// TIA Portal project "Tank_V17" (V17)

(* hardware
DEVICE "S7-1200-Station_1"  S7-1200 Station
   slot 0: "Baugruppenträger_0"  S7-1200 Rack  Rack  V1.0
   slot 1: "PLC_1"  CPU 1214C DC/DC/DC  6ES7 214-1AG40-0XB0  V4.2
   slot 3: "AQ 1x12BIT_1"  AQ1 signal board  6ES7 232-4HA30-0XB0  V1.0
*)

// ===== PLC "PLC_1"  CPU 1214C DC/DC/DC =====

VAR_GLOBAL   // PLC tag table "Standard-Variablentabelle"
   "System_Byte" AT %MB100 : Byte;
   "FirstScan" AT %M100.0 : Bool;
   "DiagStatusUpdate" AT %M100.1 : Bool;
   "AlwaysTRUE" AT %M100.2 : Bool;
   "AlwaysFALSE" AT %M100.3 : Bool;
   "Clock_Byte" AT %MB110 : Byte;
   "Clock_10Hz" AT %M110.0 : Bool;
   "Clock_5Hz" AT %M110.1 : Bool;
   "Clock_2.5Hz" AT %M110.2 : Bool;
   "Clock_2Hz" AT %M110.3 : Bool;
   "Clock_1.25Hz" AT %M110.4 : Bool;
   "Clock_1Hz" AT %M110.5 : Bool;
   "Clock_0.625Hz" AT %M110.6 : Bool;
   "Clock_0.5Hz" AT %M110.7 : Bool;
   "S0" AT %I10.0 : Bool;   // Not-Halt
   "S5-Hand" AT %I10.2 : Bool;   // Wahlschalter - Hand
   "S5-Automatik" AT %I10.3 : Bool;   // Wahlschalter - Automatik
   "S10" AT %I10.4 : Bool;   // Taster "Füllen"
   "S11" AT %I10.5 : Bool;   // Taster "Leeren"
   "S1" AT %I10.1 : Bool;   // Taster Start
   "P1" AT %Q10.0 : Bool;   // Meldeleuchte "Start"
   "P2" AT %Q10.1 : Bool;   // Meldeleuchte "Füllen"
   "P3" AT %Q10.2 : Bool;   // Meldeleuchte "Leeren"
   "B10" AT %ID40 : Real;   // Sensor Durchfluss
   "B11" AT %ID44 : Real;   // Sensor Pegel
   "P10" AT %QD40 : Real;   // Digitale Anzeige Durchfluss
   "P11" AT %QD44 : Real;   // Digitale Anzeige Pegel
   "Y1" AT %QD52 : Real;   // Füllventil
   "Y2" AT %QD56 : Real;   // Entleerventil
   "AlleAusgänge" AT %QW0 : Word;
END_VAR

FUNCTION "fc_Tank" : Void   // FC1, FBD
{ S7_Optimized_Access := 'TRUE' }
VERSION : 0.1
BEGIN

REGION Network 1: Meldeleuchte "Start"
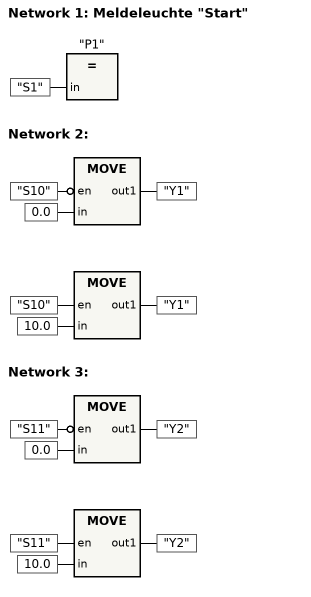
   "P1" := "S1";
END_REGION

REGION Network 2
   IF NOT "S10" THEN "Y1" := 0.0; END_IF;
   IF "S10" THEN "Y1" := 10.0; END_IF;
END_REGION

REGION Network 3
   IF NOT "S11" THEN "Y2" := 0.0; END_IF;
   IF "S11" THEN "Y2" := 10.0; END_IF;
END_REGION
END_FUNCTION

ORGANIZATION_BLOCK "Main"   // OB1, LAD, ProgramCycle
TITLE = "Main Program Sweep (Cycle)"
{ S7_Optimized_Access := 'TRUE' }
VERSION : 0.1
   VAR_INPUT
      Initial_Call : Bool;   // Initial call of this OB
      Remanence : Bool;   // =True, if remanent data are available
   END_VAR
BEGIN

REGION Network 1
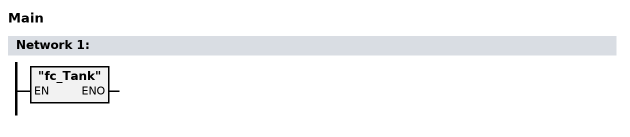
   RUNG wire#powerrail
      "fc_Tank"()
   END_RUNG
   // the same network as SCL:
   "fc_Tank"();
END_REGION
END_ORGANIZATION_BLOCK

ORGANIZATION_BLOCK "Startup"   // OB100, SCL, Startup
TITLE = "Complete Restart"
{ S7_Optimized_Access := 'TRUE' }
VERSION : 0.1
   VAR_INPUT
      LostRetentive : Bool;   // True if retentive data are lost
      LostRTC : Bool;   // True if date and time are lost
   END_VAR
BEGIN
   "AlleAusgänge" := 16#0000;
END_ORGANIZATION_BLOCK